// TIA Portal V18 export
DATA_BLOCK "man_desk_button_cell_DB"   // DB29
VERSION : 0.1
// stored: AutoNumber true, DBAccessibleFromOPCUA true, InstanceOfName _ML2_target_supplier, InstanceOfType FB
"_ML2_target_supplier"
   // VAR_INPUT
   //    ALLOWED : Bool;
   //    xServiceKey : Bool;
   //    xManButtonAny : Bool;
   //    xSwAutoCycle : Bool;
   //    xXrayCycleRuning : Bool;
   //    xGoToNextDefect : Bool;
   //    xGoToPrevDefect : Bool;
   //    xHome : Bool;
   //    xLoad : Bool;
   //    xControl1 : Bool;
   //    xControl2 : Bool;
   //    xDefectSave : Bool;
   //    xDefectsReset : Bool;
   //    Spots_pos_AR : "typeSpotList";
   //    CurPositios : "typePositions";
   //    ACK : Bool;
   //    ArrivedAll : Bool;
   //    HomePos : "typePositions";
   //    LoadPos : "typePositions";
   //    Control1Pos : "typePositions";
   //    Control2Pos : "typePositions";
   //    bSoftStop : Bool;
   // END_VAR
   // VAR_OUTPUT
   //    ExecuteAllAxisTogether : Bool;
   //    mdNotAllowed : Bool;
   //    mdServiceKey : Bool;
   //    mdCycle : Bool;
   //    mdSemi : Bool;
   //    mdMan : Bool;
   //    wsMODE : WString;
   //    wsTarget : WString;
   //    er_ws : WString;
   // END_VAR
   // VAR_IN_OUT
   //    Target_pos : "typePositions";
   //    DefectsDB : "typeDefectsDB";
   //    hmiGoToDefect : Bool;
   //    hmiGotoSpot : Bool;
   //    SPOT_i : Int;
   //    xyBeepDoneDefects : Bool;
   // END_VAR
   // VAR
   //    def_util_db { S7_SetPoint := 'True'} : "defects_util";
   //    mdSemi_was : Bool;
   //    st_goToDefectNow : Bool;
   //    q0_auto : Bool;
   //    q00_semi : Bool;
   //    q1_spot : Bool;
   //    p1_spot : Bool;
   //    q2_defect : Bool;
   //    p2_defect : Bool;
   //    q99_none : Bool;
   //    q_auto_waiting : Bool;
   //    block1 { S7_SetPoint := 'True'} : "_ML2_ts_block1";
   //    p3_home : Bool;
   //    q3_home : Bool;
   //    p4_load : Bool;
   //    q4_load : Bool;
   //    p5_control1 : Bool;
   //    q5_control1 : Bool;
   //    p6_control2 : Bool;
   //    q6_control2 : Bool;
   // END_VAR
BEGIN
END_DATA_BLOCK
